FUNCTION_BLOCK Stopped IMPLEMENTS ITF_PackMLState, ITF_States
VAR
	_MyContext : REFERENCE TO SomeMachine;
END_VAR

{warning 'add property implementation'}
PROPERTY AbortingState : ITF_PackMLState
GET
END_GET
SET
END_SET
END_PROPERTY

METHOD CyclicLogic : BOOL
VAR_INPUT
END_VAR
END_METHOD

{warning 'add method implementation '}
METHOD EStop : BOOL
END_METHOD

{warning 'add property implementation'}
PROPERTY MyNextState : ITF_PackMLState
GET
END_GET
SET
END_SET
END_PROPERTY

{warning 'add method implementation '}
METHOD Reset : BOOL
END_METHOD

{warning 'add method implementation '}
METHOD SetContext : BOOL
VAR_INPUT
	context	: REFERENCE TO SomeMachine;
END_VAR
_MyContext REF= context;
END_METHOD

{warning 'add method implementation '}
METHOD Start : BOOL
END_METHOD

{warning 'add method implementation '}
METHOD Stop : BOOL
END_METHOD

{warning 'add property implementation'}
PROPERTY StoppingState : ITF_PackMLState
GET
END_GET
SET
END_SET
END_PROPERTY

END_FUNCTION_BLOCK

(* stored: Version 1.1.0.1, ProductVersion 3.1.4024.12
   POU Stopped: Id {dc82a4e7-f66d-44be-8922-178610a55f51}, SpecialFunc None
   Property AbortingState: Id {401c6ba3-a749-4715-add0-751c1b615d6a}
   Get Get: Id {b5d3b208-5d8a-4d17-b99d-862771a4e32c}
   Set Set: Id {9daf51e6-9ac6-4b29-9932-4703d3b18521}
   Method CyclicLogic: Id {e75c9e8e-13d6-4788-9283-68c0b718b073}
   Method EStop: Id {760555aa-8dd1-4b73-8d91-d630a3bc3cb5}
   Property MyNextState: Id {94b5bce6-3d73-4d82-9eed-1017b00f2c26}
   Get Get: Id {89454a5e-64a3-46c3-9b2f-ec0bbaf27c8d}
   Set Set: Id {756f8f04-c97b-4cec-b395-e61defc80092}
   Method Reset: Id {45ca4b20-ee67-47cb-b58e-2a104fcefcc3}
   Method SetContext: Id {7016a00a-42e2-4ead-a1d6-736bd46e651a}
   Method Start: Id {20c86fab-cbe7-4b19-8451-6d5663a6fc22}
   Method Stop: Id {58229fa1-862b-4bff-b560-eaded43c244e}
   Property StoppingState: Id {79b91320-8353-4e86-b3ef-d67f712df881}
   Get Get: Id {52a36044-fdf7-4f79-8412-0aa561ff56d1}
   Set Set: Id {24e73990-bf56-4f7a-8f86-2a948b997db9} *)
